(* 
:Description: This function block represent basic TCP/IP data buffer. It is used by all TCP devices to store data to send and recive from other devices.
*)
FUNCTION_BLOCK FB_TcpBuffer

VAR CONSTANT
	iLENGTH_OF_MESSAGE		: UDINT := 8192;
	iMAX_NUMBER_OF_MESSAGES	: UDINT := 10;
END_VAR

VAR
	arrBufferMessage	: ARRAY[0..iMAX_NUMBER_OF_MESSAGES] OF ST_TcpBufferData;
	{attribute 'hide'}
	iFirstMessageIndex	: UDINT;
	{attributee 'hide'}
	iLastMessageIndex	: UDINT;
END_VAR

(* Returns TRUE if everything went fine, FALSE if buffer is full *)
METHOD MR_Append : BOOL 
VAR_INPUT
	stData	:	ST_TcpBufferData;
END_VAR
(* Clear buffer *)
IF (arrBufferMessage[iLastMessageIndex].iLength = 0) THEN
	arrBufferMessage[iLastMessageIndex] := stData;
	MR_Append := TRUE;	
	
(* Increment one index and append data to row *)
ELSIF iLastMessageIndex < iMAX_NUMBER_OF_MESSAGES THEN
	iLastMessageIndex := iLastMessageIndex + 1;
	arrBufferMessage[iLastMessageIndex] := stData;
	MR_Append := TRUE;
	
(* Start from 0 index *)
ELSIF iFirstMessageIndex > 0 THEN
	iLastMessageIndex := 0;
	arrBufferMessage[iLastMessageIndex] := stData;
	MR_Append := TRUE;

(* Buffer is full *)	
ELSE
	MR_Append := FALSE;
	
END_IF
END_METHOD

(* Clears buffer *)
METHOD MR_Clear : BOOL
VAR_INPUT
END_VAR
MEMSET(	destAddr	:=	ADR(arrBufferMessage),
		fillByte	:=	0,
		n			:=	SIZEOF(arrBufferMessage));
		
iFirstMessageIndex := 0;
iLastMessageIndex := 0;

MR_Clear := TRUE;
END_METHOD

(* Gets last data structure from buffer *)
METHOD MR_GetLast : ST_TcpBufferData
VAR_INPUT
END_VAR
MR_GetLast := arrBufferMessage[iLastMessageIndex];
END_METHOD

(* Gets last data structure from buffer and removes it*)
METHOD MR_GetNextAndRemove : ST_TcpBufferData;
VAR_INPUT
END_VAR
(*Get data *)
MR_GetNextAndRemove := arrBufferMessage[iFirstMessageIndex];

(*Remove data from index *)
MEMSET(	destAddr	:=	ADR(arrBufferMessage[iFirstMessageIndex]), 
		fillByte	:=	0, 
		n			:=	SIZEOF(arrBufferMessage[iFirstMessageIndex]));

(* Change index of first message if it's not the only message *)
IF iFirstMessageIndex <> iLastMessageIndex THEN 
	
	(* Incerment index *)
	IF iFirstMessageIndex < iMAX_NUMBER_OF_MESSAGES THEN 
		iFirstMessageIndex := iFirstMessageIndex + 1;
	
	(* End of buffer, go to 0 *)	
	ELSE 
		iFirstMessageIndex := 0;
		
	END_IF
	
END_IF
END_METHOD

END_FUNCTION_BLOCK

(* stored: Version 1.1.0.1, ProductVersion 3.1.4024.9
   POU FB_TcpBuffer: Id {289bbe3c-554e-4410-9ec9-c89a593fd113}, SpecialFunc None
   Folder Requests: Id {69451874-ffae-4a28-9201-18fd923dc5f2}
   Method MR_Append: Id {5b397181-f15d-4d43-96e8-04694368c5c1}
   Method MR_Clear: Id {4e167701-f75e-4239-bd73-356eaad0ec61}
   Method MR_GetLast: Id {14baec6b-0f2b-481e-9dfe-a4ea0507a218}
   Method MR_GetNextAndRemove: Id {a5e692dc-6490-4a88-b4e5-9412366611b6} *)
